Fanuc KAREL source: kb00106.KL

-- PROVISIONAL review KL for V1013-1; original PC SHA256 6bdb033ce5853cc3a5ef9643e5376e8bc543d8aecdc5751367ffe40c92a62375
-- Incomplete behavior may be omitted. Consult companion uncertainty JSON. Do not deploy.
PROGRAM KB00106
%NOLOCKGROUP
BEGIN
  -- UNRESOLVED_PC offsets 5-15; opcodes 27,22,31
  -- UNRESOLVED_PC offsets 20-24; opcodes 7F
END KB00106
